{attribute 'GeneratedUsingTerminal: KL9160'}
{attribute addProperty BoxType "KL9160"}
{attribute addProperty Description ""}
{attribute addProperty Physics ""}
{attribute addProperty Id "Channel_1AT %I*Channel_64AAC8C70"}
{attribute addProperty CRC "2347652594"}
{attribute addProperty Size "0"}
TYPE KL9160_8BEE55F2 :
STRUCT
	{attribute addProperty Name "Channel_1"}
	Channel_1 : Channel_64AAC8C7;
END_STRUCT
END_TYPE

(* stored: Version 1.2.0.0, ProductVersion 3.1.4024.9
   DUT KL9160_8BEE55F2: Id {ed40b6be-8d99-428f-9e08-2eb1f7383e17} *)
